PROGRAM LOCAL_COM_Controller
VAR
END_VAR

END_PROGRAM

(* stored: Version 1.1.0.1, ProductVersion 3.1.4022.18
   POU LOCAL_COM_Controller: Id {ab0f22dc-fc9a-42bd-9bd0-62af04ce36f5}, SpecialFunc None *)
